// ---- POUs/Regelungstechnik/visu/RET_VISU_Regler.TcVIS
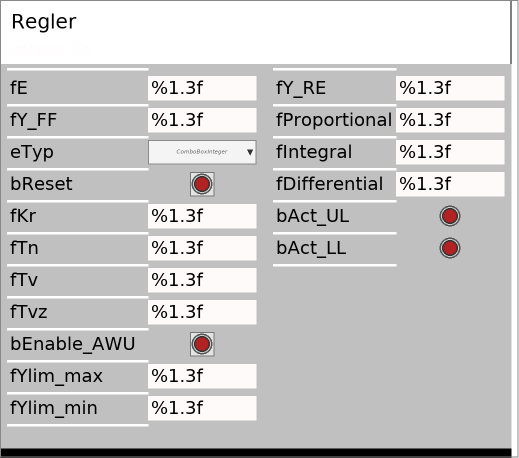
VISUALIZATION RET_VISU_Regler  // 519x458
VAR_INPUT
   {attribute 'parameterstringof' := 'm_Input_FB'}
   m_Input_INST_Str : STRING;
END_VAR
VAR_IN_OUT
   m_Input_FB : Regler;
END_VAR
    RoundedRectangle (0,0 511x81)
    RoundedRectangle (0,418 511x40)
    Rectangle (0,64 511x384)
    Lamp1 (438,204 24x24), variable: m_Input_FB.bAct_UL, style: Lamp-Lamp1-Red
    Lamp1 (438,236 24x24), variable: m_Input_FB.bAct_LL, style: Lamp-Lamp1-Red
    PushSwitch (190,172 24x24), variable: m_Input_FB.bReset, behaviour: TOGGLE, style: Switch-PushSwitch-Red
    PushSwitch (190,332 24x24), variable: m_Input_FB.bEnable_AWU, behaviour: TOGGLE, style: Switch-PushSwitch-Red
    Rectangle (8,8 511x27), "Regler"
    Rectangle (8,35 511x27), "Instance: %s", text variable: m_Input_INST_Str
    Rectangle (7,68 141x2)
    Rectangle (148,76 108x24), "%1.3f", text variable: m_Input_FB.fE
        OnMouseClick: write the text variable via Default
    Rectangle (7,76 141x24), "fE"
    Rectangle (7,104 141x2)
    Rectangle (148,108 108x24), "%1.3f", text variable: m_Input_FB.fY_FF
        OnMouseClick: write the text variable via Default
    Rectangle (7,108 141x24), "fY_FF"
    Rectangle (7,136 141x2)
    Rectangle (7,140 141x24), "eTyp"
    Rectangle (7,168 141x2)
    Rectangle (7,172 141x24), "bReset"
    Rectangle (7,200 141x2)
    Rectangle (148,204 108x24), "%1.3f", text variable: m_Input_FB.fKr
        OnMouseClick: write the text variable via Default
    Rectangle (7,204 141x24), "fKr"
    Rectangle (7,232 141x2)
    Rectangle (148,236 108x24), "%1.3f", text variable: m_Input_FB.fTn
        OnMouseClick: write the text variable via Default
    Rectangle (7,236 141x24), "fTn"
    Rectangle (7,264 141x2)
    Rectangle (148,268 108x24), "%1.3f", text variable: m_Input_FB.fTv
        OnMouseClick: write the text variable via Default
    Rectangle (7,268 141x24), "fTv"
    Rectangle (7,296 141x2)
    Rectangle (148,300 108x24), "%1.3f", text variable: m_Input_FB.fTvz
        OnMouseClick: write the text variable via Default
    Rectangle (7,300 141x24), "fTvz"
    Rectangle (7,328 141x2)
    Rectangle (7,332 141x24), "bEnable_AWU"
    Rectangle (7,360 141x2)
    Rectangle (148,364 108x24), "%1.3f", text variable: m_Input_FB.fYlim_max
        OnMouseClick: write the text variable via Default
    Rectangle (7,364 141x24), "fYlim_max"
    Rectangle (7,392 141x2)
    Rectangle (148,396 108x24), "%1.3f", text variable: m_Input_FB.fYlim_min
        OnMouseClick: write the text variable via Default
    Rectangle (7,396 141x24), "fYlim_min"
    Rectangle (7,424 141x2)
    Rectangle (273,68 123x2)
    Rectangle (396,76 108x24), "%1.3f", text variable: m_Input_FB.fY_RE
    Rectangle (273,76 123x24), "fY_RE"
    Rectangle (273,104 123x2)
    Rectangle (396,108 108x24), "%1.3f", text variable: m_Input_FB.fProportional
    Rectangle (273,108 123x24), "fProportional"
    Rectangle (273,136 123x2)
    Rectangle (396,140 108x24), "%1.3f", text variable: m_Input_FB.fIntegral
    Rectangle (273,140 123x24), "fIntegral"
    Rectangle (273,168 123x2)
    Rectangle (396,172 108x24), "%1.3f", text variable: m_Input_FB.fDifferential
    Rectangle (273,172 123x24), "fDifferential"
    Rectangle (273,200 123x2)
    Rectangle (273,204 123x24), "bAct_UL"
    Rectangle (273,232 123x2)
    Rectangle (273,236 123x24), "bAct_LL"
    Rectangle (273,264 123x2)
    Frame (148,140 108x24), input disabled if: False
        shows VISU_HELPER_Combobox_eReglertyp(varEnum := m_Input_FB.eTyp)
END_VISUALIZATION

// ---- POUs/Regelungstechnik/visu/RET_VISU_Signalgenerator.TcVIS
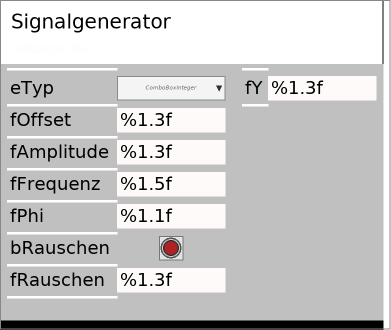
VISUALIZATION RET_VISU_Signalgenerator  // 391x330
VAR_INPUT
   {attribute 'parameterstringof' := 'm_Input_FB'}
   m_Input_INST_Str : STRING;
END_VAR
VAR_IN_OUT
   m_Input_FB : Signalgenerator;
END_VAR
    RoundedRectangle (0,0 383x81)
    RoundedRectangle (0,290 383x40)
    Rectangle (0,64 383x256)
    PushSwitch (159,236 24x24), variable: m_Input_FB.bRauschen, behaviour: TOGGLE, style: Switch-PushSwitch-Red
    Rectangle (8,8 383x27), "Signalgenerator"
    Rectangle (8,35 383x27), "Instance: %s", text variable: m_Input_INST_Str
    Rectangle (7,68 110x2)
    Rectangle (7,76 110x24), "eTyp"
    Rectangle (7,104 110x2)
    Rectangle (117,108 108x24), "%1.3f", text variable: m_Input_FB.fOffset
        OnMouseClick: write the text variable via Default
    Rectangle (7,108 110x24), "fOffset"
    Rectangle (7,136 110x2)
    Rectangle (117,140 108x24), "%1.3f", text variable: m_Input_FB.fAmplitude
        OnMouseClick: write the text variable via Default
    Rectangle (7,140 110x24), "fAmplitude"
    Rectangle (7,168 110x2)
    Rectangle (117,172 108x24), "%1.5f", text variable: m_Input_FB.fFrequenz
        OnMouseClick: write the text variable via Default
    Rectangle (7,172 110x24), "fFrequenz"
    Rectangle (7,200 110x2)
    Rectangle (117,204 108x24), "%1.1f", text variable: m_Input_FB.fPhi
        OnMouseClick: write the text variable via Default
    Rectangle (7,204 110x24), "fPhi"
    Rectangle (7,232 110x2)
    Rectangle (7,236 110x24), "bRauschen"
    Rectangle (7,264 110x2)
    Rectangle (117,268 108x24), "%1.3f", text variable: m_Input_FB.fRauschen
        OnMouseClick: write the text variable via Default
    Rectangle (7,268 110x24), "fRauschen"
    Rectangle (7,296 110x2)
    Rectangle (242,68 26x2)
    Rectangle (268,76 108x24), "%1.3f", text variable: m_Input_FB.fY
    Rectangle (242,76 26x24), "fY"
    Rectangle (242,104 26x2)
    Frame (117,76 108x24), input disabled if: False
        shows VISU_HELPER_Combobox_eSignalform(varEnum := m_Input_FB.eTyp)
END_VISUALIZATION

// ---- POUs/Regelungstechnik/visu/RET_VISU_Strecke.TcVIS
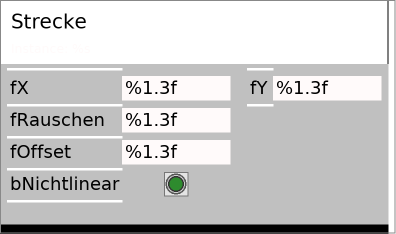
VISUALIZATION RET_VISU_Strecke  // 396x234
VAR_INPUT
   {attribute 'parameterstringof' := 'm_Input_FB'}
   m_Input_INST_Str : STRING;
END_VAR
VAR_IN_OUT
   m_Input_FB : Strecke;
END_VAR
    RoundedRectangle (0,0 388x81)
    RoundedRectangle (0,194 388x40)
    Rectangle (0,64 388x160)
    PushSwitch (164,172 24x24), variable: m_Input_FB.bNichtlinear, behaviour: TOGGLE, style: Switch-PushSwitch-Green
    Rectangle (8,8 388x27), "Strecke"
    Rectangle (8,35 388x27), "Instance: %s", text variable: m_Input_INST_Str
    Rectangle (7,68 115x2)
    Rectangle (122,76 108x24), "%1.3f", text variable: m_Input_FB.fX
        OnMouseClick: write the text variable via Default
    Rectangle (7,76 115x24), "fX"
    Rectangle (7,104 115x2)
    Rectangle (122,108 108x24), "%1.3f", text variable: m_Input_FB.fRauschen
        OnMouseClick: write the text variable via Default
    Rectangle (7,108 115x24), "fRauschen"
    Rectangle (7,136 115x2)
    Rectangle (122,140 108x24), "%1.3f", text variable: m_Input_FB.fOffset
        OnMouseClick: write the text variable via Default
    Rectangle (7,140 115x24), "fOffset"
    Rectangle (7,168 115x2)
    Rectangle (7,172 115x24), "bNichtlinear"
    Rectangle (7,200 115x2)
    Rectangle (247,68 26x2)
    Rectangle (273,76 108x24), "%1.3f", text variable: m_Input_FB.fY
    Rectangle (247,76 26x24), "fY"
    Rectangle (247,104 26x2)
END_VISUALIZATION

// ---- POUs/Regelungstechnik/visu/TextListForCombobox_eReglertyp.TcTLO
TEXTLIST TextListForCombobox_eReglertyp
  1 = 'P'
  2 = 'I'
  3 = 'PI'
  4 = 'PDT1'
  5 = 'PIDT1'
   = ''
END_TEXTLIST

// ---- POUs/Regelungstechnik/visu/TextListForCombobox_eSignalform.TcTLO
TEXTLIST TextListForCombobox_eSignalform
  1 = 'OFF'
  2 = 'OFFSET'
  3 = 'RECHTECK'
  4 = 'DREIECK'
  5 = 'SINUS'
   = ''
END_TEXTLIST

// ---- POUs/Regelungstechnik/visu/VISU_HELPER_Combobox_eReglertyp.TcVIS
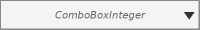
VISUALIZATION VISU_HELPER_Combobox_eReglertyp  // 200x30
VAR_IN_OUT
    varEnum : eReglertyp;
END_VAR
    ComboBoxInteger (0,0 200x30), variable: varEnum, text list: 'TextListForCombobox_eReglertyp'
END_VISUALIZATION

// ---- POUs/Regelungstechnik/visu/VISU_HELPER_Combobox_eSignalform.TcVIS
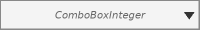
VISUALIZATION VISU_HELPER_Combobox_eSignalform  // 200x30
VAR_IN_OUT
    varEnum : eReglertyp;
END_VAR
    ComboBoxInteger (0,0 200x30), variable: varEnum, text list: 'TextListForCombobox_eSignalform'
END_VISUALIZATION

// ---- VISUs/Achse_R.TcVIS
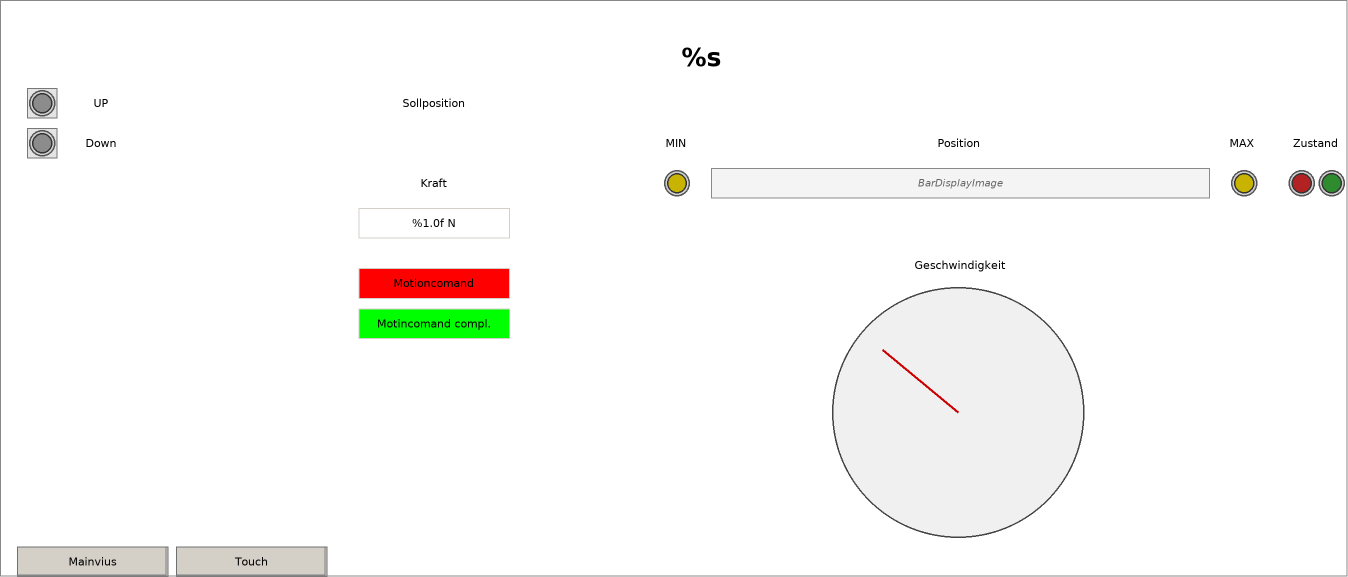
VISUALIZATION Achse_R  // 1348x577
    Frame (6,8 1342x569)
        shows Visu_Achse(Axis := MAIN.Axis_R)
END_VISUALIZATION

// ---- VISUs/Achse_S.TcVIS
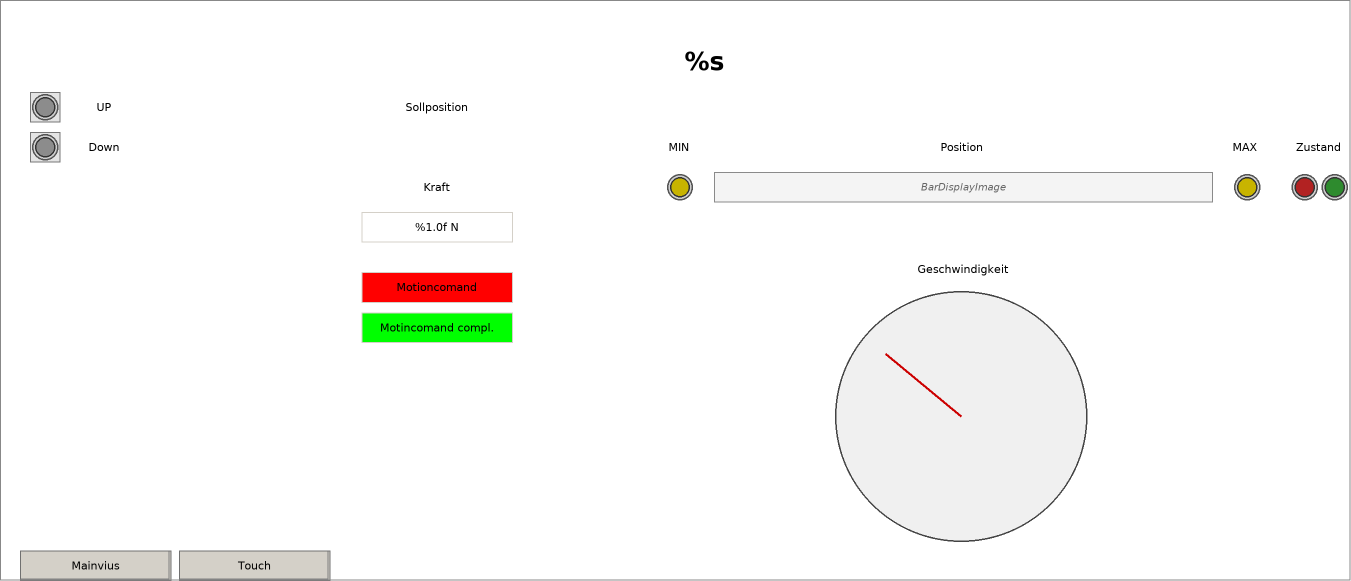
VISUALIZATION Achse_S  // 1351x581
    Frame (9,12 1342x569)
        shows Visu_Achse(Axis := MAIN.Axis_S)
END_VISUALIZATION

// ---- VISUs/Achse_T.TcVIS
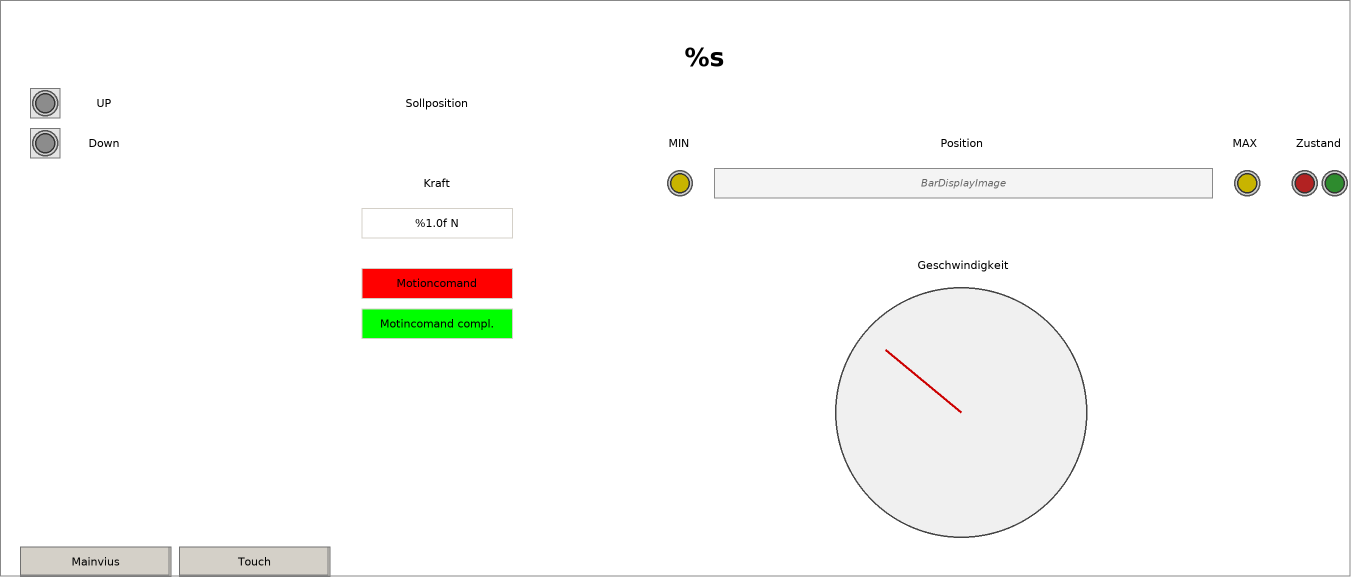
VISUALIZATION Achse_T  // 1351x577
    Frame (9,8 1342x569)
        shows Visu_Achse(Axis := MAIN.Axis_T)
END_VISUALIZATION

// ---- VISUs/FigureGeneratorDisplay.TcVIS
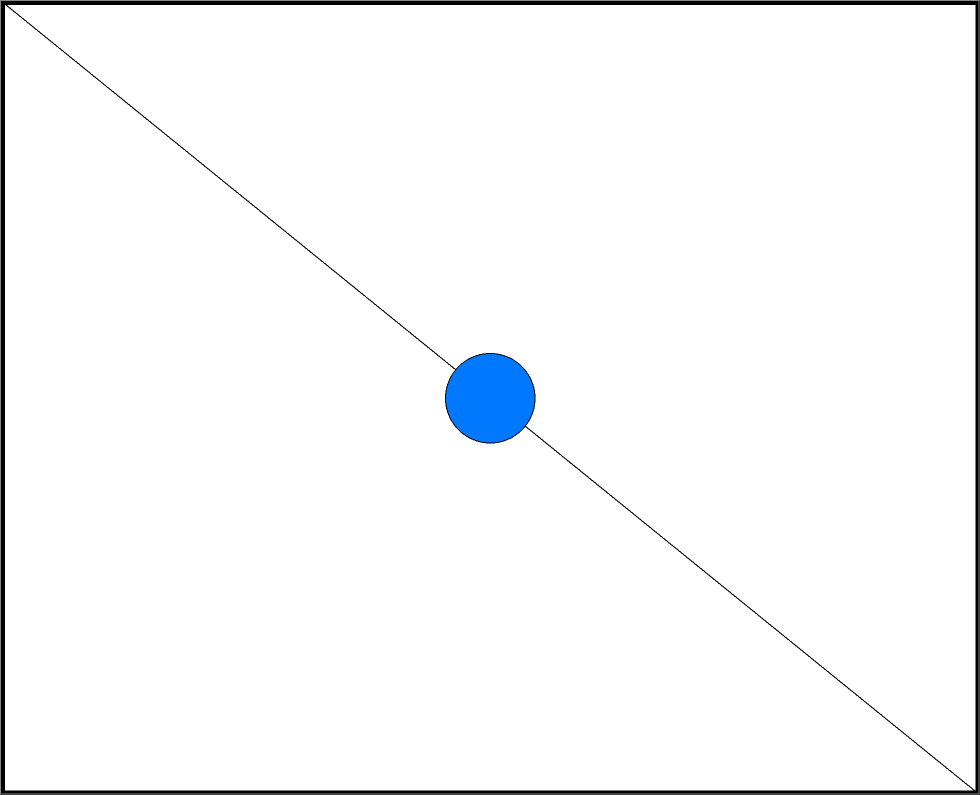
VISUALIZATION FigureGeneratorDisplay  // 980x795
    Rectangle (0,0 980x795)
    Frame (0,0 980x795)
        shows Polygon(pVisu := MAIN.FB_FigureGenerator.pVisu, VisuLenght := MAIN.FB_FigureGenerator.VisuLenght)
    Ellipse (445,353 90x90), invisible if: NOT Touchpanel.bContactAvailable
        p3560616238: Touchpanel.touch_scale_x.rX_mm*2.5
        p2738717112: -Touchpanel.touch_scale_y.rX_mm*2.5
END_VISUALIZATION

// ---- VISUs/Home.TcVIS
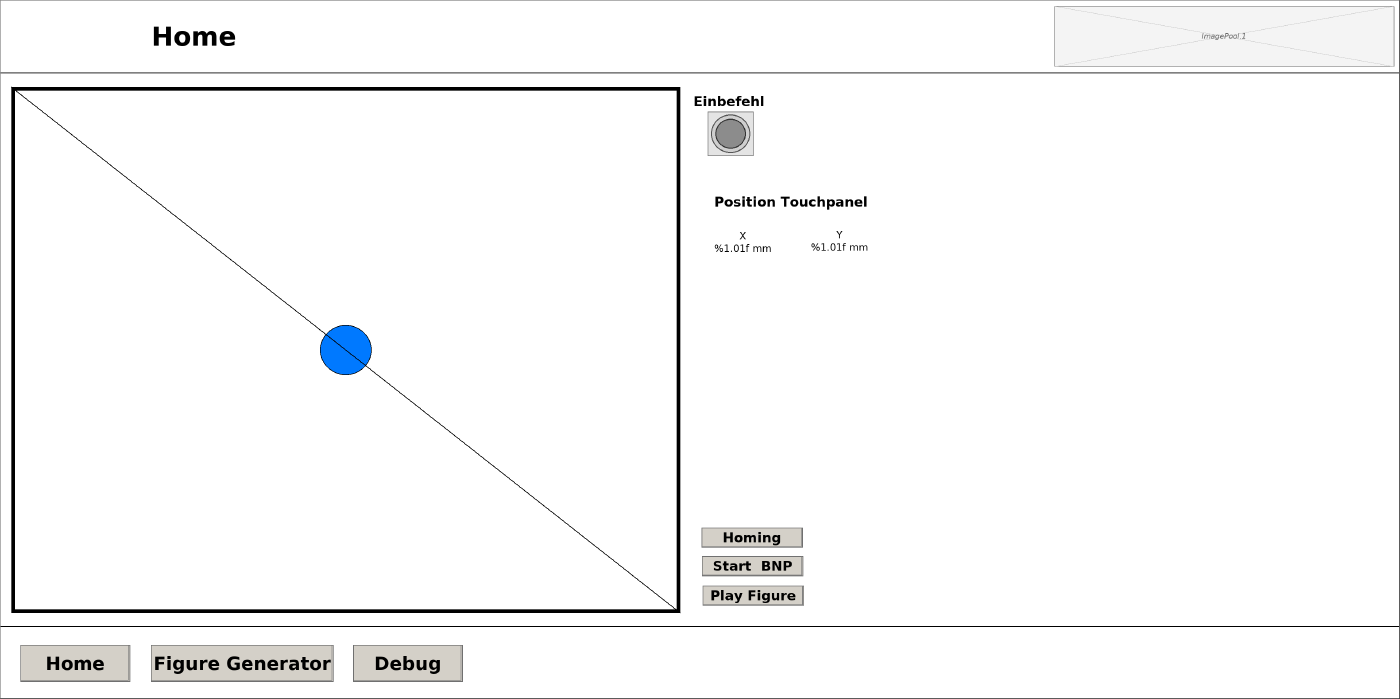
VISUALIZATION Home  // 1919x959
    Rectangle (0,0 1919x910)
    Rectangle (0,0 1919x100)
    Rectangle (0,859 1919x100)
    Button (28,885 150x50), "Home"
    Label (191,25 150x50), "Home"
    Image (1445,8 466x83), image: ImagePool.1
    Button (207,885 250x50), "Figure Generator"
        OnMouseClick: change screen: FigureGenerator1
    Button (484,885 150x50), "Debug"
        OnMouseClick: change screen: Debug
    Frame (12,116 1205x725)
        shows FigurePlayer()
END_VISUALIZATION

// ---- VISUs/FigureGenerator1.TcVIS
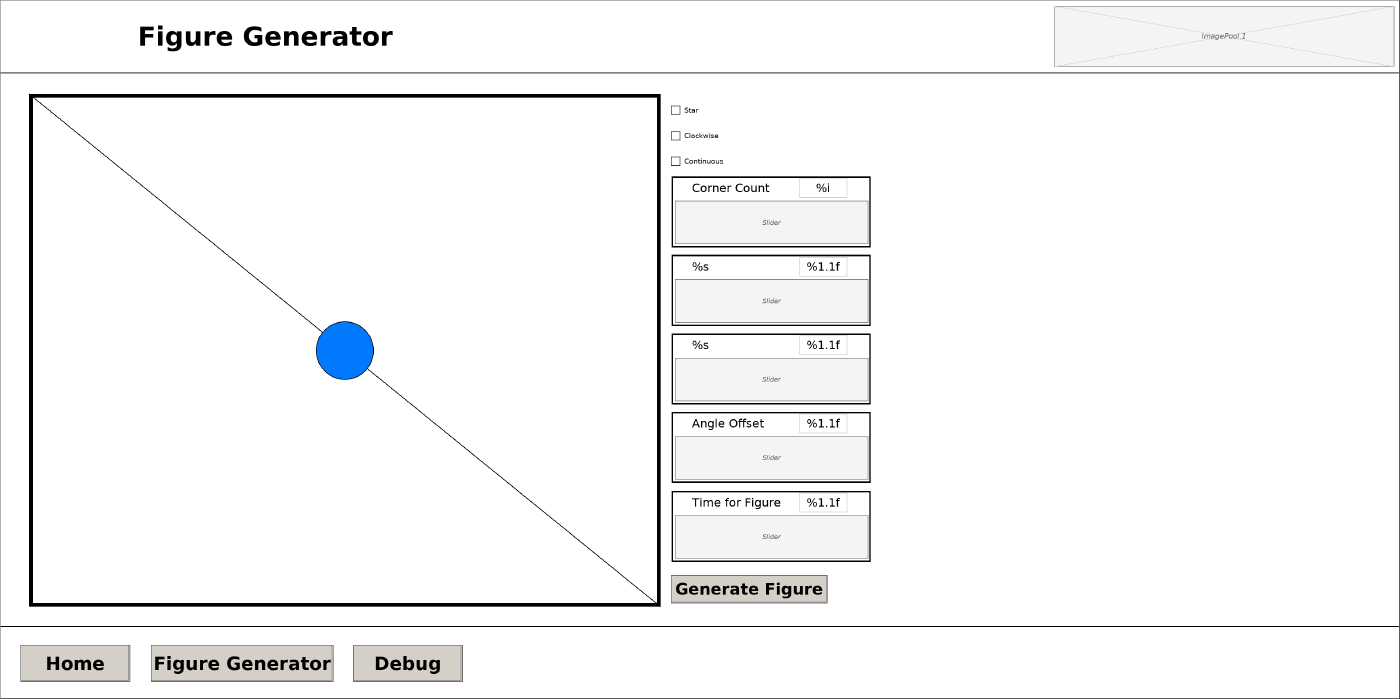
VISUALIZATION FigureGenerator1  // 1919x959
    Rectangle (0,0 1919x910)
    Rectangle (0,0 1919x100)
    Rectangle (0,859 1919x100)
    Button (28,885 150x50), "Home"
        OnMouseClick: change screen: Home
    Label (193,25 342x50), "Figure Generator"
    Image (1445,8 466x83), image: ImagePool.1
    Button (207,885 250x50), "Figure Generator"
    Button (484,885 150x50), "Debug"
        OnMouseClick: change screen: Debug
    Frame (36,125 1157x707)
        shows FigureGenerator()
END_VISUALIZATION

// ---- VISUs/Debug.TcVIS
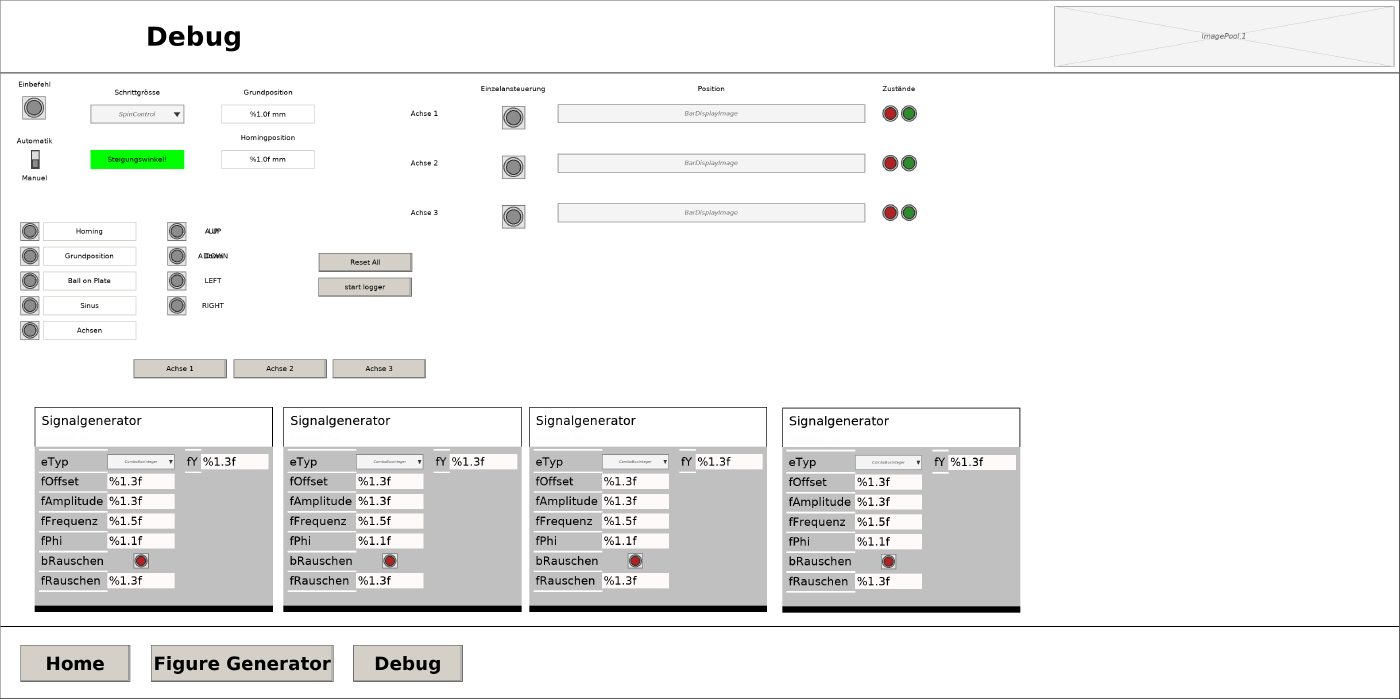
VISUALIZATION Debug  // 1919x959
    Rectangle (0,0 1919x910)
    Rectangle (0,0 1919x100)
    Rectangle (0,859 1919x100)
    Button (28,885 150x50), "Home"
        OnMouseClick: change screen: Home
    Label (191,25 150x50), "Debug"
    Image (1445,8 466x83), image: ImagePool.1
    Button (207,885 250x50), "Figure Generator"
        OnMouseClick: change screen: FigureGenerator1
    Button (484,885 150x50), "Debug"
    Frame (8,93 1397x747)
        shows Mainvisu()
END_VISUALIZATION

// ---- VISUs/InputNumSlider_Corner.TcVIS
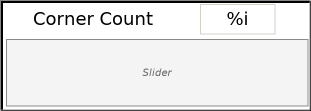
VISUALIZATION InputNumSlider_Corner  // 311x111
    Rectangle (1,1 310x110)
    Label (30,4 150x30), "Corner Count"
    Textfield (200,4 75x30), "%i", text variable: MAIN.FB_FigureGenerator.nCornerCountInp
        OnMouseClick: write the text variable via Default, min 3, max 100
    Slider (6,39 302x67), variable: MAIN.FB_FigureGenerator.nCornerCountInp, scale 3..13
END_VISUALIZATION

// ---- VISUs/InputNumSlider_Radius.TcVIS
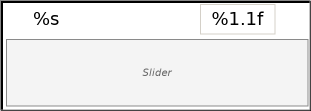
VISUALIZATION InputNumSlider_Radius  // 311x111
VAR_IN_OUT
number : REAL;
name : STRING;
END_VAR
    Rectangle (1,1 310x110)
    Slider (6,39 302x67), variable: number, scale 0..180
    Textfield (30,4 150x30), "%s", text variable: name
    Textfield (200,4 75x30), "%1.1f", text variable: number
        OnMouseClick: write the text variable via Default, min 0, max 180
END_VISUALIZATION

// ---- VISUs/InputNumSlider_Angle.TcVIS
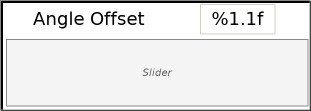
VISUALIZATION InputNumSlider_Angle  // 311x111
VAR_IN_OUT
number : REAL;
END_VAR
    Rectangle (1,1 310x110)
    Slider (6,39 302x67), variable: number, scale 0..360
    Textfield (30,4 150x30), "Angle Offset"
    Textfield (200,4 75x30), "%1.1f", text variable: number
        OnMouseClick: write the text variable via Default, min 0, max 360
END_VISUALIZATION

// ---- VISUs/InputNumSlider_Time.TcVIS
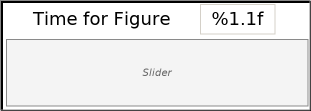
VISUALIZATION InputNumSlider_Time  // 311x111
VAR_IN_OUT
number : REAL;
END_VAR
    Rectangle (1,1 310x110)
    Slider (6,39 302x67), variable: number, scale 0..100
    Textfield (30,4 150x30), "Time for Figure"
    Textfield (200,4 75x30), "%1.1f", text variable: number
        OnMouseClick: write the text variable via Default, min 0, max 360
END_VISUALIZATION

// ---- VISUs/Mainvisu.TcVIS
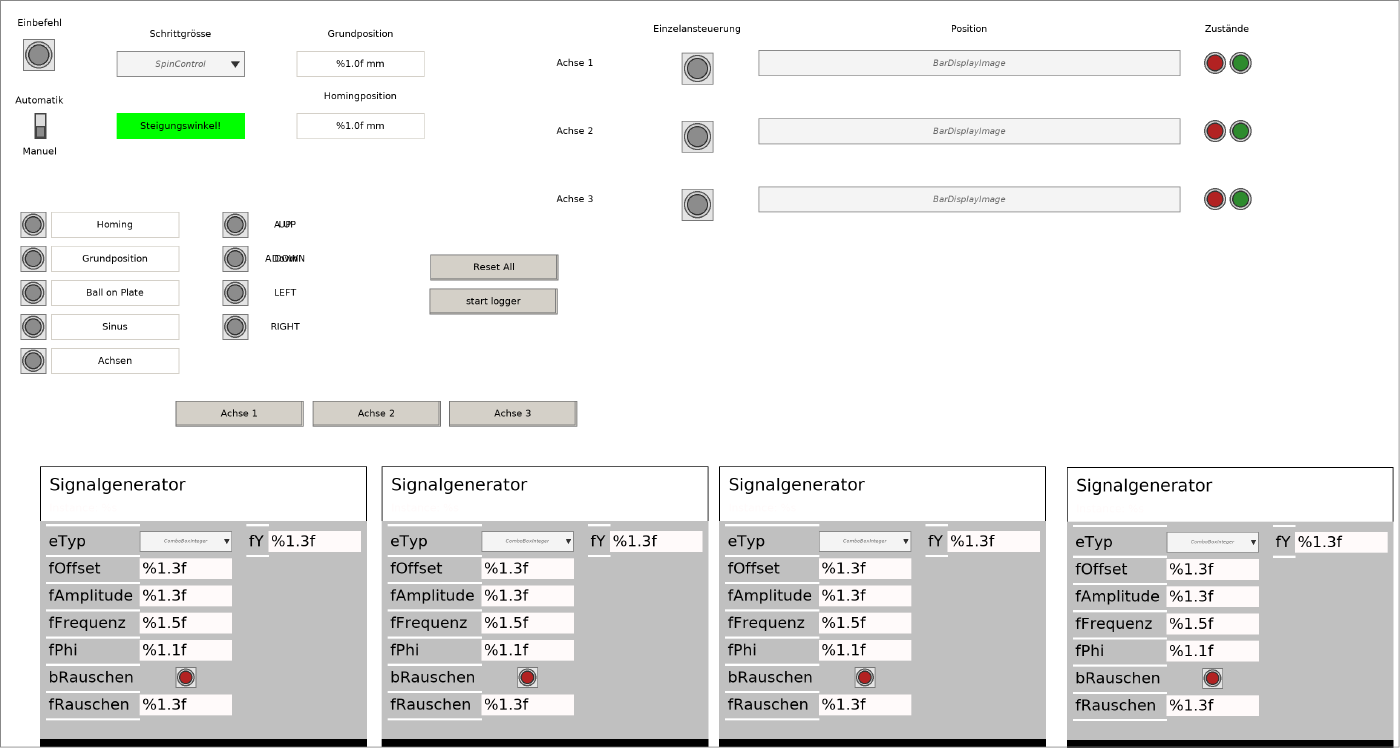
VISUALIZATION Mainvisu  // 1643x879
    DipSwitch (32,133 31x30), variable: GVL.Automatik, behaviour: TOGGLE, style: Switch-DipSwitch-Gray
    Label (12,103 69x30), "Automatik"
    Label (12,163 69x30), "Manuel"
    PushSwitch (260,249 32x30), variable: GVL.UP, invisible if: GVL.Achsenkontrolle, behaviour: TAP, style: Switch-PushSwitch-Gray
    PushSwitch (260,289 32x30), variable: GVL.Down, invisible if: GVL.Achsenkontrolle, behaviour: TAP, style: Switch-PushSwitch-Gray
    Label (300,249 69x30), "UP", invisible if: GVL.Achsenkontrolle
    Label (300,289 69x30), "Down", invisible if: GVL.Achsenkontrolle
    Label (348,25 150x30), "Grundposition"
    PushSwitch (22,289 34x30), variable: GVL.Grundposition, behaviour: TAP, style: Switch-PushSwitch-Gray
    Textfield (348,60 150x30), "%1.0f mm", text variable: GVL.Eingabe_Sollposition
    Label (348,98 150x30), "Homingposition"
    Textfield (348,133 150x30), "%1.0f mm", text variable: GVL.Eingabe_Grundposition
    Label (12,12 69x30), "Einbefehl"
    SpinControl (137,60 150x30), variable: GVL.StepSize
    Label (137,25 150x30), "Schrittgrösse"
    BarDisplayImage (890,59 495x30), value: MAIN.Axis_R.ActualPosition, style: BarDisplayImage-Gray, scale format: %.0f, scale 0..200
    Label (890,19 495x30), "Position"
    BarDisplayImage (890,139 495x30), value: MAIN.Axis_S.ActualPosition, style: BarDisplayImage-Gray, scale format: %.0f, scale 0..200
    BarDisplayImage (890,219 495x30), value: MAIN.Axis_T.ActualPosition, style: BarDisplayImage-Gray, scale format: %.0f, scale 0..200
    Lamp1 (1410,59 32x30), variable: MAIN.Axis_R.WarningActive, style: Lamp-Lamp1-Red
    Lamp1 (1410,139 32x30), variable: MAIN.Axis_S.WarningActive, style: Lamp-Lamp1-Red
    Lamp1 (1410,219 32x30), variable: MAIN.Axis_T.WarningActive, style: Lamp-Lamp1-Red
    Lamp1 (1440,59 32x30), variable: MAIN.Axis_R.Ready, style: Lamp-Lamp1-Green
    Lamp1 (1440,139 32x30), variable: MAIN.Axis_S.Ready, style: Lamp-Lamp1-Green
    Lamp1 (1440,219 32x30), variable: MAIN.Axis_T.Ready, style: Lamp-Lamp1-Green
    PushSwitchLed (800,59 37x43), variable: MAIN.Axis_R.bManual, behaviour: TOGGLE, style: Switch-PushSwitchLed-Gray
    PushSwitchLed (800,139 37x43), variable: MAIN.Axis_S.bManual, behaviour: TOGGLE, style: Switch-PushSwitchLed-Gray
    PushSwitchLed (800,219 37x43), variable: MAIN.Axis_T.bManual, behaviour: TOGGLE, style: Switch-PushSwitchLed-Gray
    Label (743,19 150x30), "Einzelansteuerung"
    PushSwitchLed (27,43 37x43), variable: gvl.Einbefehl, behaviour: TOGGLE, style: Switch-PushSwitchLed-Gray
    PushSwitch (22,329 34x30), variable: GVL.BndP, behaviour: TAP, style: Switch-PushSwitch-Gray
    Textfield (60,329 150x30), "Ball on Plate", colour toggle: MAIN.Modus = Mode.BallundPlate
        toggle GVL.BndP
    PushSwitch (22,369 34x30), variable: GVL.Sinus, behaviour: TAP, style: Switch-PushSwitch-Gray
    Textfield (60,369 150x30), "Sinus", colour toggle: MAIN.Modus = Mode.Sinus
        toggle GVL.BndP
    Textfield (60,289 150x30), "Grundposition", colour toggle: MAIN.Modus = Mode.Position
        toggle GVL.BndP
    Textfield (137,133 150x30), "Steigungswinkel!", colour toggle: GVL.Warnung_Steigungswinkel
        toggle GVL.BndP
    PushSwitch (260,249 32x30), variable: GVL.XAchseUp, invisible if: not GVL.Achsenkontrolle, behaviour: TAP, style: Switch-PushSwitch-Gray
    PushSwitch (260,289 32x30), variable: GVL.XAchseDown, invisible if: not GVL.Achsenkontrolle, behaviour: TAP, style: Switch-PushSwitch-Gray
    Label (300,249 69x30), "A UP", invisible if: not GVL.Achsenkontrolle
    Label (300,289 69x30), "A DOWN", invisible if: not GVL.Achsenkontrolle
    PushSwitch (260,329 32x30), variable: GVL.YAchseDown, invisible if: not GVL.Achsenkontrolle, behaviour: TAP, style: Switch-PushSwitch-Gray
    PushSwitch (260,369 32x30), variable: GVL.YAchseUp, invisible if: not GVL.Achsenkontrolle, behaviour: TAP, style: Switch-PushSwitch-Gray
    Label (300,329 69x30), "LEFT", invisible if: not GVL.Achsenkontrolle
    Label (300,369 69x30), "RIGHT", invisible if: not GVL.Achsenkontrolle
    Textfield (60,409 150x30), "Achsen", colour toggle: MAIN.Modus = Mode.Tilt
    PushSwitch (22,249 34x30), variable: GVL.Homing, behaviour: TAP, style: Switch-PushSwitch-Gray
    Textfield (60,249 150x30), "Homing", colour toggle: MAIN.Modus = Mode.Homing
        toggle GVL.BndP
    PushSwitch (22,409 34x30), variable: GVL.Tilt, behaviour: TAP, style: Switch-PushSwitch-Gray
    Label (600,59 150x30), "Achse 1"
    Label (600,139 150x30), "Achse 2"
    Label (600,219 150x30), "Achse 3"
    Label (1410,19 60x30), "Zustände"
    Button (206,471 150x30), "Achse 1"
        OnMouseDown: change screen: Achse_R
    Button (367,471 150x30), "Achse 2"
        OnMouseDown: change screen: Achse_S
    Button (527,471 150x30), "Achse 3"
        OnMouseDown: change screen: Achse_T
    Button (505,299 150x30), "Reset All"
        tap GVL.reset
    Frame (47,548 391x330)
        shows RET_VISU_Signalgenerator(m_Input_FB := CONTROLLER.fbSignalgeno_Y_x)
    Frame (448,548 391x330)
        shows RET_VISU_Signalgenerator(m_Input_FB := CONTROLLER.fbSignalgeno_Y_y)
    Frame (844,548 391x330)
        shows RET_VISU_Signalgenerator(m_Input_FB := CONTROLLER.fbSignalgeno_W_x)
    Frame (1252,549 391x330)
        shows RET_VISU_Signalgenerator(m_Input_FB := CONTROLLER.fbSignalgeno_W_y)
    Button (504,339 150x30), "start logger", pressed state: CONTROLLER.bLoggerRunning
        OnMouseDown: toggle CONTROLLER.bLoggerRunning
END_VISUALIZATION

// ---- VISUs/Polygon.TcVIS
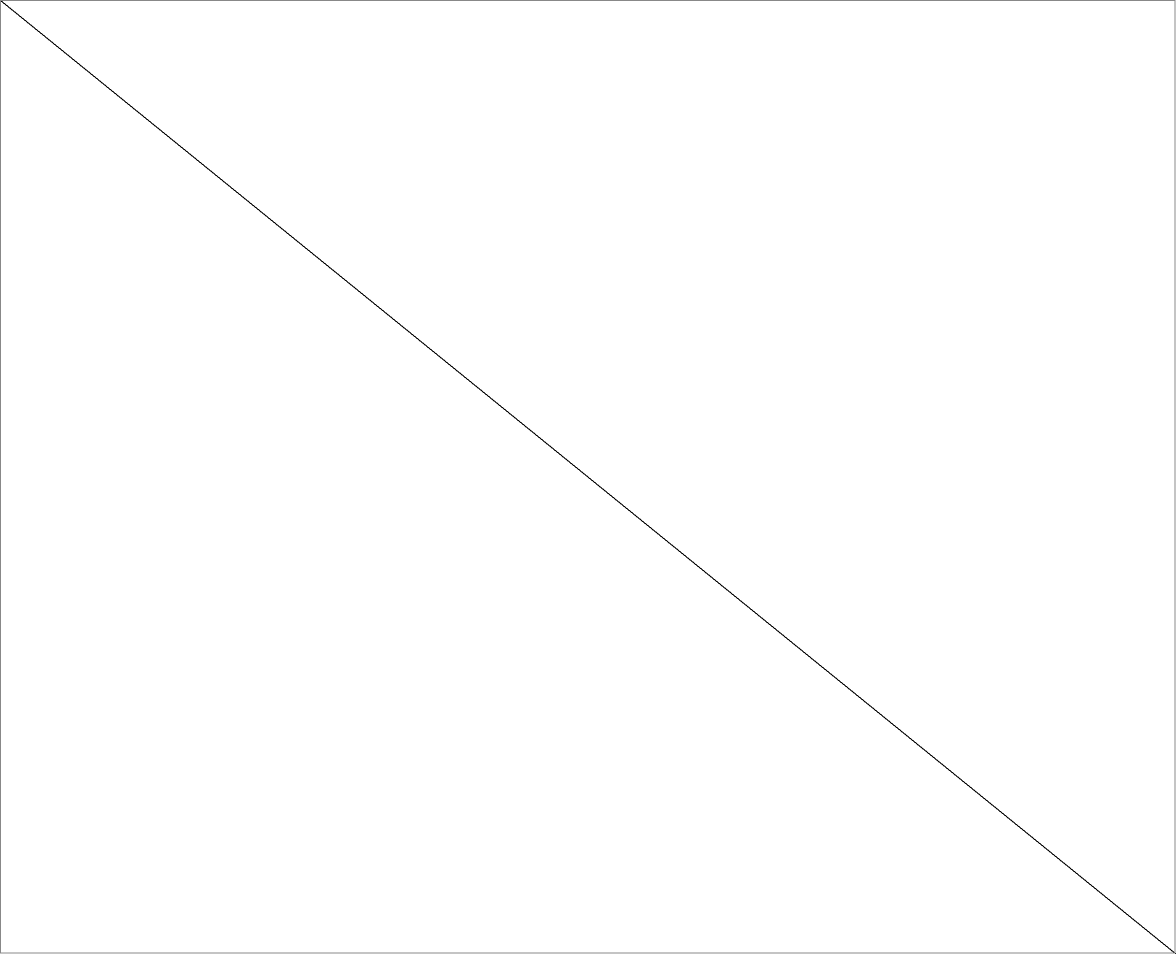
VISUALIZATION Polygon  // 1176x954
VAR_IN_OUT
	pVisu : POINTER TO ARRAY[0..999] OF VisuElems.VisuStructPoint;
	VisuLenght : INT;
END_VAR
    Polyline (0,0) (1176,954) (0,0) (0,0) (0,0)
        p1285906596: pVisu
        p3184209983: VisuLenght
END_VISUALIZATION

// ---- VISUs/FigurePlayer.TcVIS
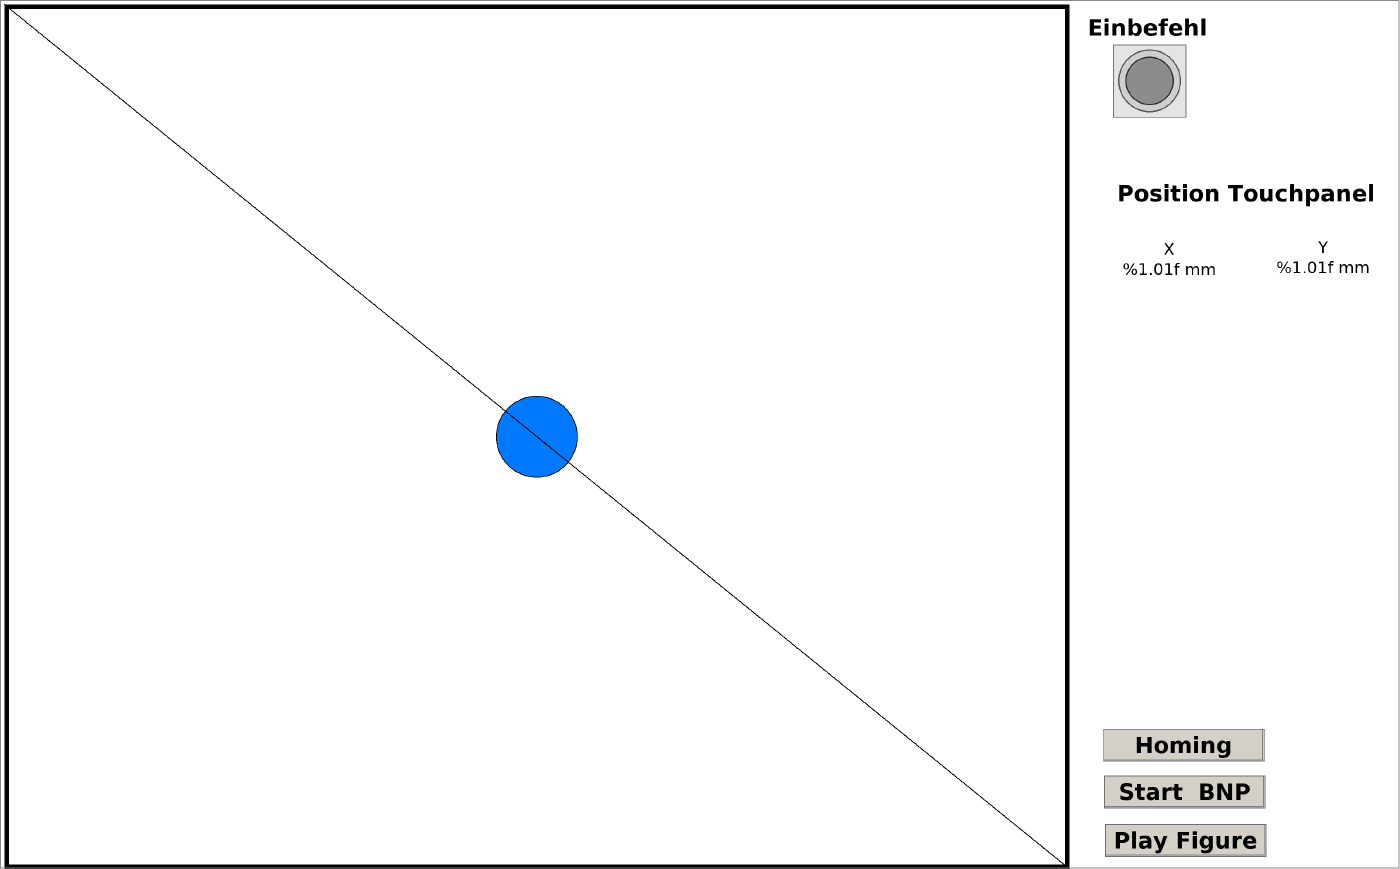
VISUALIZATION FigurePlayer  // 1557x967
    Rectangle (1386,261 171x51), "Y %1.01f mm", text variable: Touchpanel.touch_scale_y.rX_mm
    Rectangle (1215,263 171x51), "X %1.01f mm", text variable: Touchpanel.touch_scale_x.rX_mm
    Label (1215,185 342x60), "Position Touchpanel"
    Frame (5,5 1184x962)
        shows FigurePlayerDisplay()
    Button (1229,917 179x36), "Play Figure", pressed state: CONTROLLER.FB_FigurePlayer_0.bStart
        toggle CONTROLLER.FB_FigurePlayer_0.bStart
    Label (1200,11 152x39), "Einbefehl"
    PushSwitchLed (1238,49 81x82), variable: gvl.Einbefehl, behaviour: TOGGLE, style: Switch-PushSwitchLed-Gray
    Button (1228,863 179x36), "Start BNP", pressed state: GVL.BNP_Aktiv
        tap GVL.BndP
    Button (1227,811 179x36), "Homing", pressed state: GVL.Homing
        tap GVL.Homing
END_VISUALIZATION

// ---- VISUs/FigureGenerator.TcVIS
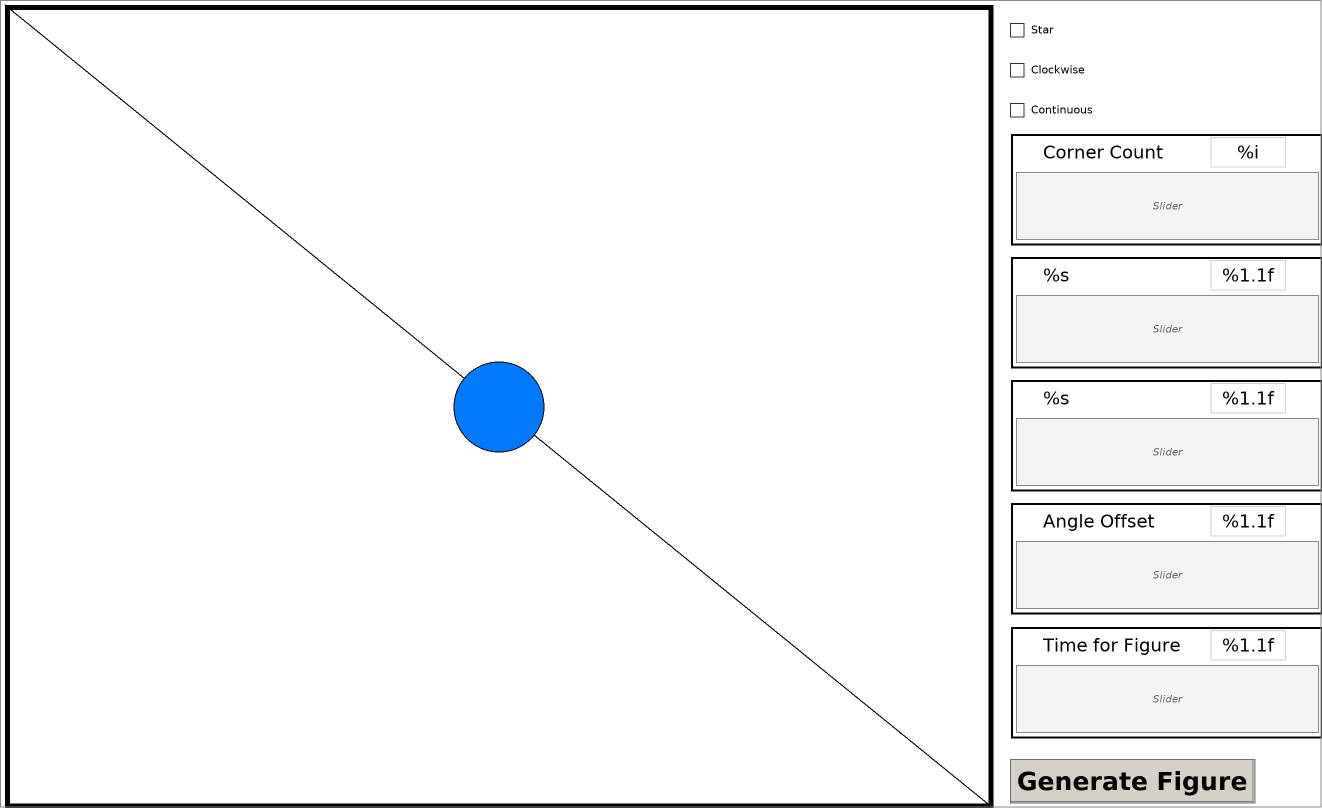
VISUALIZATION FigureGenerator  // 1322x808
    Checkbox (1008,15 150x30), "Star", variable: MAIN.FB_FigureGenerator.bStar
    Checkbox (1008,95 150x30), "Continuous", variable: MAIN.FB_FigureGenerator.bContinus
    Button (1010,759 245x44), "Generate Figure", pressed state: MAIN.FB_FigureGenerator.bGenerate
        tap MAIN.FB_FigureGenerator.bGenerate
    Frame (1010,133 312x112)
        shows InputNumSlider_Corner()
    Frame (1010,256 312x112)
        shows InputNumSlider_Radius(number := MAIN.FB_FigureGenerator.rRadius1, name := MAIN.FB_FigureGenerator.sRadius1)
    Frame (1010,379 312x112)
        shows InputNumSlider_Radius(number := MAIN.FB_FigureGenerator.rRadius2, name := MAIN.FB_FigureGenerator.sRadius2)
    Frame (1010,502 312x112)
        shows InputNumSlider_Angle(number := MAIN.FB_FigureGenerator.rAngleOffset)
    Frame (1010,626 312x112)
        shows InputNumSlider_Time(number := MAIN.FB_FigureGenerator.rFigureTime)
    Checkbox (1008,55 150x30), "Clockwise", variable: MAIN.FB_FigureGenerator.bClockwise
    Frame (5,5 988x803)
        shows FigureGeneratorDisplay()
END_VISUALIZATION

// ---- VISUs/FigurePlayerDisplay.TcVIS
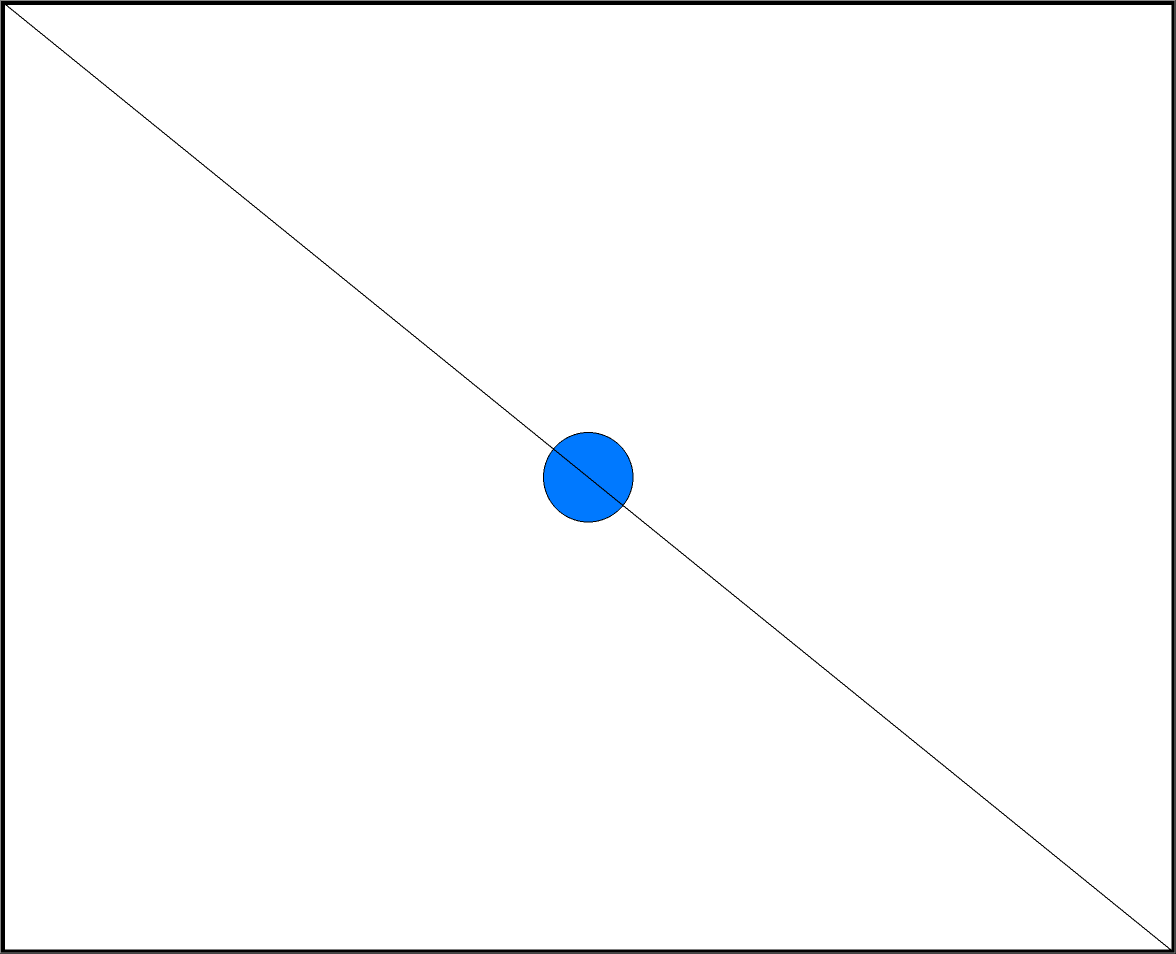
VISUALIZATION FigurePlayerDisplay  // 1176x954
    Rectangle (0,0 1176x954)
    Ellipse (543,432 90x90), invisible if: NOT Touchpanel.bContactAvailable
        p3560616238: Touchpanel.touch_scale_x.rX_mm*3
        p2738717112: -Touchpanel.touch_scale_y.rX_mm*3
    Frame (0,0 1176x954)
        shows Polygon(pVisu := CONTROLLER.FB_FigurePlayer_0.pFigure^.pVisu, VisuLenght := CONTROLLER.FB_FigurePlayer_0.pFigure^.VisuLenght)
    Frame (0,0 1176x954)
        shows Polygon_1(pVisu := MAIN.FB_BallTrack.pVisu, VisuLenght := MAIN.FB_BallTrack.VisuLenght)
END_VISUALIZATION

// ---- VISUs/Polygon_1.TcVIS
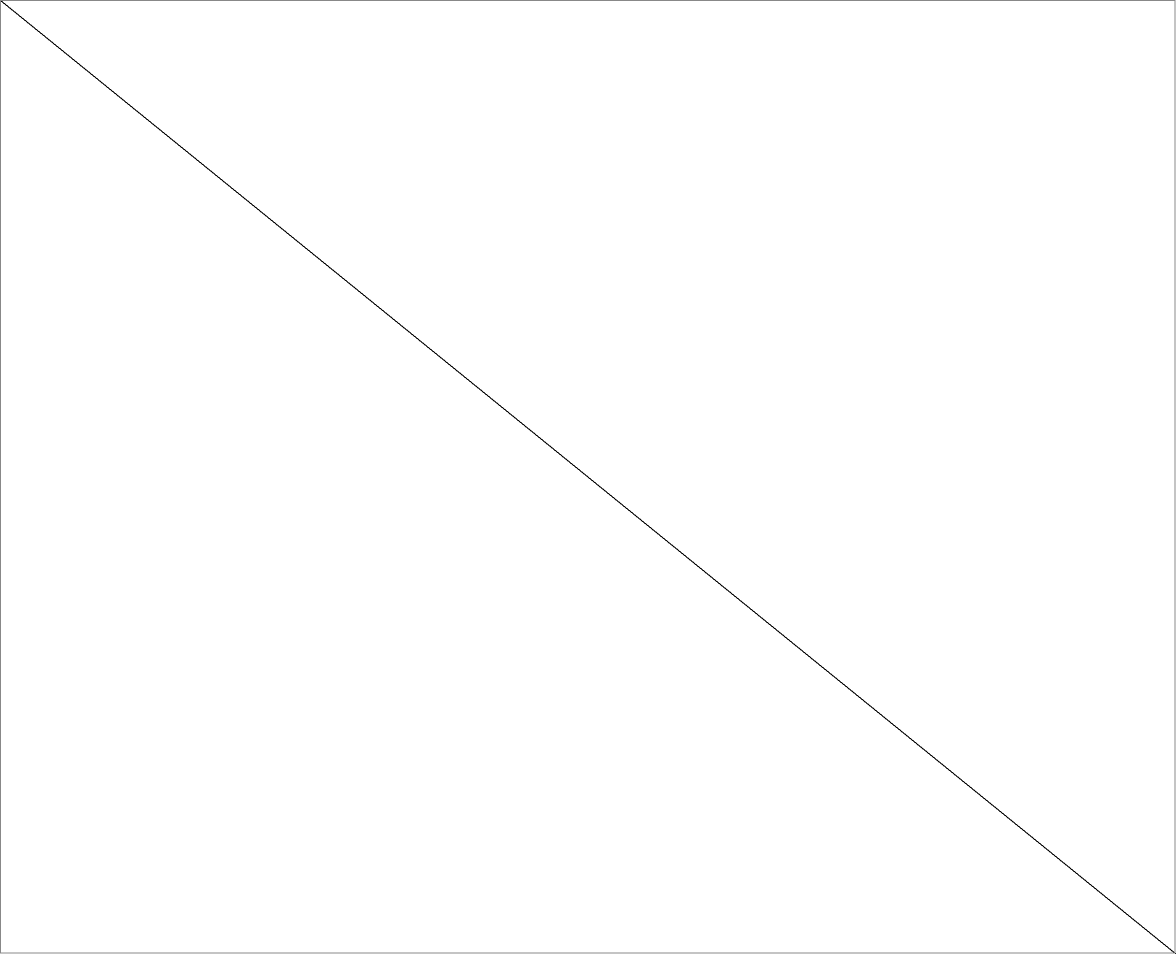
VISUALIZATION Polygon_1  // 1176x954
VAR_IN_OUT
	pVisu : POINTER TO ARRAY[0..999] OF VisuElems.VisuStructPoint;
	VisuLenght : INT;
END_VAR
    Polyline (0,0) (1176,954) (0,0) (0,0) (0,0)
        p1285906596: pVisu
        p3184209983: VisuLenght
END_VISUALIZATION

// ---- VISUs/Visu_Achse.TcVIS
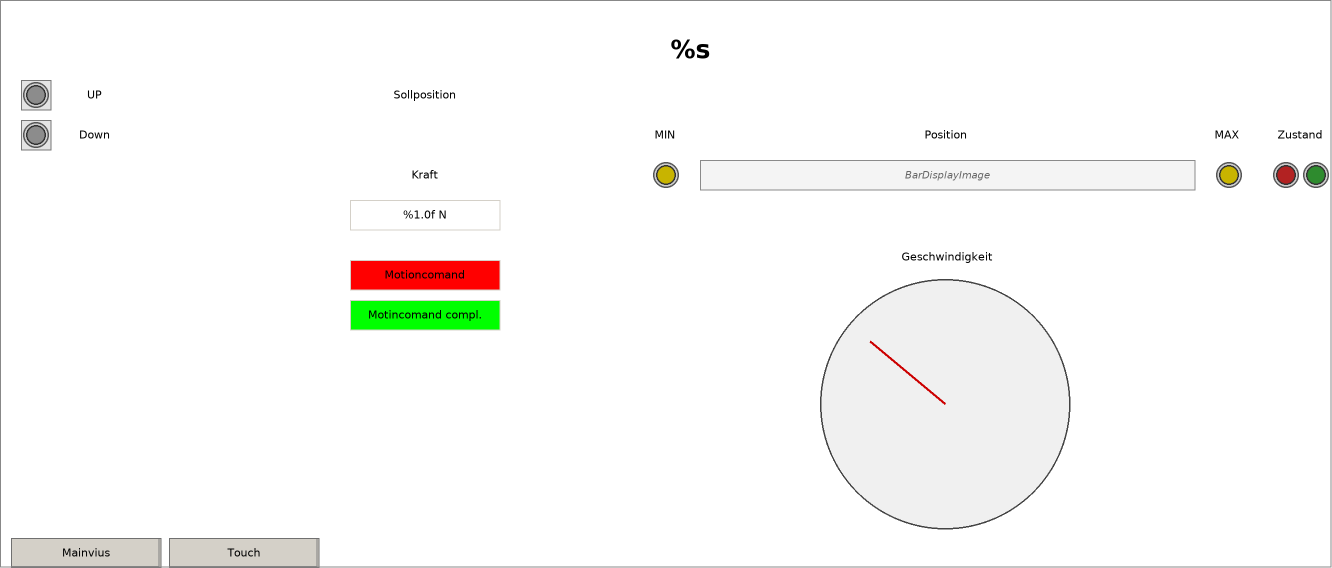
VISUALIZATION Visu_Achse  // 1332x568
VAR_IN_OUT
	Axis :FBCylTronicCylinder;
END_VAR
    Label (700,120 495x30), "Position"
    PushSwitch (20,80 32x30), variable: Axis.bUP, invisible if: NOT Axis.bManual or GVL.Achsenkontrolle, behaviour: TAP, style: Switch-PushSwitch-Gray
    PushSwitch (20,120 32x30), variable: Axis.bDOWN, invisible if: NOT Axis.bManual or GVL.Achsenkontrolle, behaviour: TAP, style: Switch-PushSwitch-Gray
    Label (60,80 69x30), "UP", invisible if: NOT Axis.bManual or GVL.Achsenkontrolle
    Label (60,120 69x30), "Down", invisible if: NOT Axis.bManual or GVL.Achsenkontrolle
    Label (350,80 150x30), "Sollposition"
    BarDisplayImage (700,160 495x30), value: Axis.ActualPosition, style: BarDisplayImage-Gray, scale format: %.0f, scale 0..200
    Lamp1 (1270,160 32x30), variable: Axis.WarningActive, style: Lamp-Lamp1-Red
    Lamp1 (1300,160 32x30), variable: Axis.Ready, style: Lamp-Lamp1-Green
    Label (350,160 150x30), "Kraft"
    Textfield (350,200 150x30), "%1.0f N", text variable: Axis.ActualForce
    Label (872,242 150x30), "Geschwindigkeit"
    Meter360 (820,279 250x250), value: Axis.ActualSpeed, style: Meter-Meter360-Gray, scale format: %.0f, scale -220..220
    Lamp1 (650,160 32x30), variable: Axis.LimitSwitchIn, style: Lamp-Lamp1-Yellow
    Lamp1 (1213,160 32x30), variable: Axis.LimitSwitchOut, style: Lamp-Lamp1-Yellow
    Textfield (350,300 150x30), "Motincomand compl.", invisible if: NOT Axis.MotionCommandCompleted
    Textfield (350,260 150x30), "Motioncomand", invisible if: NOT Axis.MotionModeActive
    Label (635,120 60x30), "MIN"
    Label (1197,120 60x30), "MAX"
    Label (1270,120 60x30), "Zustand"
    Button (11,538 150x30), "Mainvius"
        OnMouseDown: change screen: Mainvisu
    Button (169,538 150x30), "Touch"
        OnMouseDown: change screen: FigurePlayer
    Textfield (297,12 787x74), "%s", text variable: Axis.stAxisName
END_VISUALIZATION
